// TIA Portal V19 export
TYPE "LAF_typeDiagnosticsSimple"
TITLE = LAF_typeDiagnosticsSimple
// Diagnostics data type template simplified
// stored: Access Published
   STRUCT
      status { ExternalVisible := 'False'; ExternalWritable := 'False'} : Word;   // Status of the Block or error identification when error occurred
      subfunctionStatus { ExternalVisible := 'False'; ExternalWritable := 'False'} : Word;   // Status or return value of called FB's, FCs and system blocks
   END_STRUCT;
END_TYPE
